FUNCTION_BLOCK UNPK_BYTE (* Unpacks a BYTE to 8 BOOLs *)
  (* Standard: 61499-1; Classification: Math *)
  (* Version 0.1, 2007-04-02, JHC, Holobloc Inc, Corrected type of IN. *)
  (* Version 0.0, 2002-05-07, JHC, Rockwell Automation, Copied/modified from UNPK_WORD. *)
  (* Compiler header: package fb.rt.math; *)
  (* Compiler Java IBM VisualAge 3.0 *)
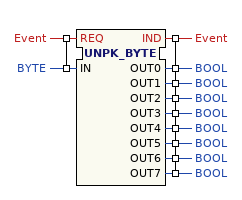
  EVENT_INPUT
    REQ WITH IN; (* Unpack Request *)
  END_EVENT
  EVENT_OUTPUT
    IND WITH OUT0, OUT1, OUT2, OUT3, OUT4, OUT5, OUT6, OUT7; (* Data Change Notification *)
  END_EVENT
  VAR_INPUT
    IN : BYTE; (* Data to Unpack *)
  END_VAR
  VAR_OUTPUT
    OUT0 : BOOL; (* Unpacked Data *)
    OUT1 : BOOL;
    OUT2 : BOOL;
    OUT3 : BOOL;
    OUT4 : BOOL;
    OUT5 : BOOL;
    OUT6 : BOOL;
    OUT7 : BOOL;
  END_VAR
  SERVICE APPLICATION/PACK_WORD
    SEQUENCE dataChanged
      APPLICATION.REQ(IN) -> PACK_WORD.unpack() -> APPLICATION.IND(OUT0,...,OUT7);
    END_SEQUENCE
    SEQUENCE dataUnchanged
      APPLICATION.REQ(IN) -> PACK_WORD.unpack();
    END_SEQUENCE
  END_SERVICE
END_FUNCTION_BLOCK
